// TIA Portal V19 export
FUNCTION "A0302_Bordatrice_RegolazioneFormato_OB1_CALL" : Void   // FC151, LAD
// stored: SetENOAutomatically false
   VAR_TEMP
      RETVAL_SET_CINT : Int;
      Check_Low : Bool;
      ChecK_High : Bool;
   END_VAR
   VAR_TEMP   // added for the SCL form of the ladder/FBD networks
      _w1 : Bool;
      _w2 : Bool;
      _w3 : Bool;
   END_VAR
BEGIN

REGION Network 2
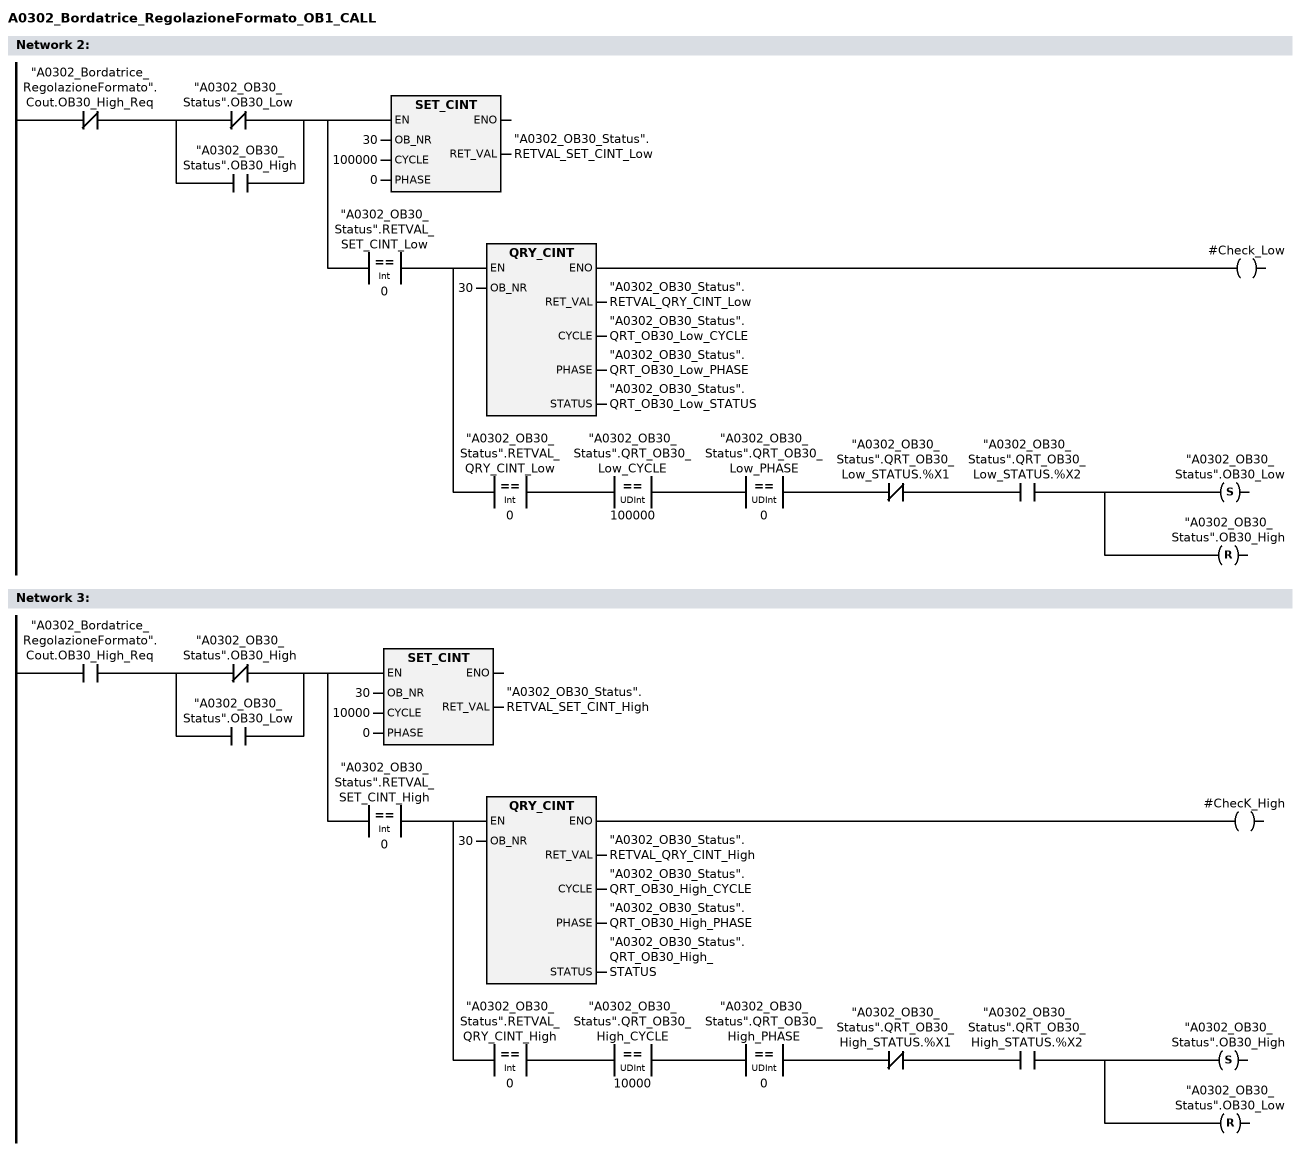
   RUNG wire#powerrail
      I_Contact( "A0302_Bordatrice_RegolazioneFormato".Cout.OB30_High_Req )
      wire#w1
      I_Contact( "A0302_OB30_Status".OB30_Low )
      wire#w2
      SET_CINT(OB_NR := 30, CYCLE := 100000, PHASE := 0, RET_VAL => "A0302_OB30_Status".RETVAL_SET_CINT_Low)
   END_RUNG
   RUNG wire#w1
      Contact( "A0302_OB30_Status".OB30_High )
   END_RUNG wire#w2
   RUNG wire#w2
      { S7_Templates := "SrcType := Int" } EQ_Contact(in1 := "A0302_OB30_Status".RETVAL_SET_CINT_Low, in2 := 0)
      wire#w3
      QRY_CINT(OB_NR := 30, RET_VAL => "A0302_OB30_Status".RETVAL_QRY_CINT_Low, CYCLE => "A0302_OB30_Status".QRT_OB30_Low_CYCLE, PHASE => "A0302_OB30_Status".QRT_OB30_Low_PHASE, STATUS => "A0302_OB30_Status".QRT_OB30_Low_STATUS)
      Coil( #Check_Low )
   END_RUNG
   RUNG wire#w3
      { S7_Templates := "SrcType := Int" } EQ_Contact(in1 := "A0302_OB30_Status".RETVAL_QRY_CINT_Low, in2 := 0)
      { S7_Templates := "SrcType := UDInt" } EQ_Contact(in1 := "A0302_OB30_Status".QRT_OB30_Low_CYCLE, in2 := 100000)
      { S7_Templates := "SrcType := UDInt" } EQ_Contact(in1 := "A0302_OB30_Status".QRT_OB30_Low_PHASE, in2 := 0)
      I_Contact( "A0302_OB30_Status".QRT_OB30_Low_STATUS.%X1 )
      Contact( "A0302_OB30_Status".QRT_OB30_Low_STATUS.%X2 )
      wire#w4
      S_Coil( "A0302_OB30_Status".OB30_Low )
   END_RUNG
   RUNG wire#w4
      R_Coil( "A0302_OB30_Status".OB30_High )
   END_RUNG
   // the same network as SCL:
   #_w1 := NOT "A0302_Bordatrice_RegolazioneFormato".Cout.OB30_High_Req AND (NOT "A0302_OB30_Status".OB30_Low OR "A0302_OB30_Status".OB30_High);
   IF #_w1 THEN
       "A0302_OB30_Status".RETVAL_SET_CINT_Low := SET_CINT(OB_NR := 30, CYCLE := 100000, PHASE := 0);
   END_IF;
   #_w2 := #_w1 AND ("A0302_OB30_Status".RETVAL_SET_CINT_Low = 0);
   "A0302_OB30_Status".RETVAL_QRY_CINT_Low := QRY_CINT(EN := #_w2,
                           OB_NR := 30,
                           CYCLE => "A0302_OB30_Status".QRT_OB30_Low_CYCLE,
                           PHASE => "A0302_OB30_Status".QRT_OB30_Low_PHASE,
                           STATUS => "A0302_OB30_Status".QRT_OB30_Low_STATUS,
                           ENO => #_w3);
   #Check_Low := #_w3;
   IF #_w2 AND ("A0302_OB30_Status".RETVAL_QRY_CINT_Low = 0) AND ("A0302_OB30_Status".QRT_OB30_Low_CYCLE = 100000) AND ("A0302_OB30_Status".QRT_OB30_Low_PHASE = 0) AND NOT "A0302_OB30_Status".QRT_OB30_Low_STATUS.%X1 AND "A0302_OB30_Status".QRT_OB30_Low_STATUS.%X2 THEN
       "A0302_OB30_Status".OB30_Low := TRUE;
       "A0302_OB30_Status".OB30_High := FALSE;
   END_IF;
END_REGION

REGION Network 3
   RUNG wire#powerrail
      Contact( "A0302_Bordatrice_RegolazioneFormato".Cout.OB30_High_Req )
      wire#w1
      I_Contact( "A0302_OB30_Status".OB30_High )
      wire#w2
      SET_CINT(OB_NR := 30, CYCLE := 10000, PHASE := 0, RET_VAL => "A0302_OB30_Status".RETVAL_SET_CINT_High)
   END_RUNG
   RUNG wire#w1
      Contact( "A0302_OB30_Status".OB30_Low )
   END_RUNG wire#w2
   RUNG wire#w2
      { S7_Templates := "SrcType := Int" } EQ_Contact(in1 := "A0302_OB30_Status".RETVAL_SET_CINT_High, in2 := 0)
      wire#w3
      QRY_CINT(OB_NR := 30, RET_VAL => "A0302_OB30_Status".RETVAL_QRY_CINT_High, CYCLE => "A0302_OB30_Status".QRT_OB30_High_CYCLE, PHASE => "A0302_OB30_Status".QRT_OB30_High_PHASE, STATUS => "A0302_OB30_Status".QRT_OB30_High_STATUS)
      Coil( #ChecK_High )
   END_RUNG
   RUNG wire#w3
      { S7_Templates := "SrcType := Int" } EQ_Contact(in1 := "A0302_OB30_Status".RETVAL_QRY_CINT_High, in2 := 0)
      { S7_Templates := "SrcType := UDInt" } EQ_Contact(in1 := "A0302_OB30_Status".QRT_OB30_High_CYCLE, in2 := 10000)
      { S7_Templates := "SrcType := UDInt" } EQ_Contact(in1 := "A0302_OB30_Status".QRT_OB30_High_PHASE, in2 := 0)
      I_Contact( "A0302_OB30_Status".QRT_OB30_High_STATUS.%X1 )
      Contact( "A0302_OB30_Status".QRT_OB30_High_STATUS.%X2 )
      wire#w4
      S_Coil( "A0302_OB30_Status".OB30_High )
   END_RUNG
   RUNG wire#w4
      R_Coil( "A0302_OB30_Status".OB30_Low )
   END_RUNG
   // the same network as SCL:
   #_w1 := "A0302_Bordatrice_RegolazioneFormato".Cout.OB30_High_Req AND (NOT "A0302_OB30_Status".OB30_High OR "A0302_OB30_Status".OB30_Low);
   IF #_w1 THEN
       "A0302_OB30_Status".RETVAL_SET_CINT_High := SET_CINT(OB_NR := 30, CYCLE := 10000, PHASE := 0);
   END_IF;
   #_w2 := #_w1 AND ("A0302_OB30_Status".RETVAL_SET_CINT_High = 0);
   "A0302_OB30_Status".RETVAL_QRY_CINT_High := QRY_CINT(EN := #_w2,
                           OB_NR := 30,
                           CYCLE => "A0302_OB30_Status".QRT_OB30_High_CYCLE,
                           PHASE => "A0302_OB30_Status".QRT_OB30_High_PHASE,
                           STATUS => "A0302_OB30_Status".QRT_OB30_High_STATUS,
                           ENO => #_w3);
   #ChecK_High := #_w3;
   IF #_w2 AND ("A0302_OB30_Status".RETVAL_QRY_CINT_High = 0) AND ("A0302_OB30_Status".QRT_OB30_High_CYCLE = 10000) AND ("A0302_OB30_Status".QRT_OB30_High_PHASE = 0) AND NOT "A0302_OB30_Status".QRT_OB30_High_STATUS.%X1 AND "A0302_OB30_Status".QRT_OB30_High_STATUS.%X2 THEN
       "A0302_OB30_Status".OB30_High := TRUE;
       "A0302_OB30_Status".OB30_Low := FALSE;
   END_IF;
END_REGION
END_FUNCTION
